(* PLC project Unnamed, Unknown Unnamed 1 *)
(* stored: creationDateTime 2025-10-22T19:37:31, modificationDateTime 2025-10-29T13:50:30 *)

PROGRAM plc_controller
  VAR
    In_Start_Stop AT %IX100.2 : BOOL;
    In_Temp_Up AT %IX100.0 : BOOL;
    In_Temp_Down AT %IX100.1 : BOOL;
    In_Emergency_Stop AT %IX100.3 : BOOL;
    Out_Status_LED AT %QX100.7 : BOOL;
    Out_Display_LED0 AT %QX100.6 : BOOL;
    Out_Display_LED1 AT %QX100.5 : BOOL;
    Out_Display_LED2 AT %QX100.4 : BOOL;
    Out_Display_LED3 AT %QX100.3 : BOOL;
    Out_Display_LED4 AT %QX100.2 : BOOL;
    Out_Display_LED5 AT %QX100.1 : BOOL;
  END_VAR
  VAR
    Out_Servo_PWM_Chann : SINT := 1;
    Servo_Freq : REAL := 50.0;
    Servo_Angle : REAL := 0.0;
    Heating_On : BOOL := FALSE;
    Element_On : BOOL := FALSE;
    Emergency_Stop : BOOL;
    Global_Enable : BOOL;
    Display_Index : INT := 0;
    Temp_Setting : INT := 0;
    Temperature : REAL;
    MAX_TEMP_SETTING : INT := 10;  (* CONSTANT describes the maximum temperature setting *)
    R_TRIG0 : R_TRIG;
    CTUD0 : CTUD;
    TON0 : TON;
    R_TRIG1 : R_TRIG;
    CTUD1 : CTUD;
    PID0 : PID;
    TON1 : TON;
    R_TRIG2 : R_TRIG;
    R_TRIG3 : R_TRIG;
  END_VAR
  VAR  (* added by the conversion: wires and edge detectors of the diagram *)
    _NOT21_OUT : BOOL;
    R_TRIG1_2 : R_TRIG;
    R_TRIG2_2 : R_TRIG;
    R_TRIG3_2 : R_TRIG;
    R_TRIG4 : R_TRIG;
    _MUL240_OUT : REAL;
  END_VAR

(* FBD diagram, written out as Structured Text *)
(* Heating on/off toggle functionality *)
(* Simple heating simulation *)
(* Multiply counter output, and add room temperature. *)
(* Emergency Stop *)
(* Temperature setting controls *)
(* Change display index in set mode *)
_NOT21_OUT := NOT Heating_On;
R_TRIG1_2(CLK := NOT CTUD0.QU AND In_Temp_Up AND _NOT21_OUT);
R_TRIG2_2(CLK := In_Temp_Down AND _NOT21_OUT AND NOT CTUD0.QD);
CTUD0(CU := R_TRIG1_2.Q, CD := R_TRIG2_2.Q, PV := MAX_TEMP_SETTING);
Temp_Setting := CTUD0.CV;
R_TRIG0(CLK := In_Start_Stop);
Heating_On := (R_TRIG0.Q XOR Heating_On) AND Global_Enable;
Out_Status_LED := Heating_On;
(* Change display index in set heating mode *)
(* Display temperature setting *)
Out_Display_LED0 := Display_Index = 0 OR Display_Index = 1;
Out_Display_LED3 := Display_Index = 5 OR Display_Index = 6 OR Display_Index = 7;
(* PID Control Loop
- P = -0.5
- I = 1000.0
- D = 0.5 *)
Out_Display_LED1 := Display_Index = 1 OR Display_Index = 2 OR Display_Index = 3;
Out_Display_LED4 := Display_Index = 7 OR Display_Index = 8 OR Display_Index = 9;
Out_Display_LED2 := Display_Index = 3 OR Display_Index = 4 OR Display_Index = 5;
Out_Display_LED5 := Display_Index = 9 OR Display_Index = 10;
TON0(IN := NOT R_TRIG1.Q, PT := T#20ms);
R_TRIG1(CLK := TON0.Q);
R_TRIG3_2(CLK := R_TRIG1.Q AND Element_On);
R_TRIG4(CLK := NOT Element_On AND R_TRIG1.Q);
CTUD1(CU := R_TRIG3_2.Q, CD := R_TRIG4.Q, PV := 1000);
Temperature := INT_TO_REAL(CTUD1.CV) * 0.1 + 60.0;
IF Global_Enable AND NOT Heating_On THEN Display_Index := Temp_Setting; END_IF;
IF Heating_On THEN Display_Index := LIMIT(0, REAL_TO_INT((Temperature - 80.0) / 100.0 * INT_TO_REAL(MAX_TEMP_SETTING)), MAX_TEMP_SETTING); END_IF;
PID0(AUTO := TRUE, PV := Temperature, SP := INT_TO_REAL(Temp_Setting * 10 + 80), KP := -0.5, TR := 1000.0, TD := 0.5, CYCLE := T#20ms);
Element_On := Heating_On AND REAL_TO_BOOL(LIMIT(0.0, PID0.XOUT, 1.0));
(* Servo valve controls
CHANNEL = 0 for %QW0
FREQ = 50Hz *)
TON1(IN := NOT R_TRIG2.Q, PT := T#100ms);
R_TRIG2(CLK := TON1.Q);
IF R_TRIG2.Q THEN Servo_Angle := LIMIT(0.0, SEL(NOT Heating_On, Servo_Angle + 1.8, Servo_Angle - 1.8), 144.0); END_IF;
R_TRIG3(CLK := In_Emergency_Stop);
Emergency_Stop := R_TRIG3.Q XOR Emergency_Stop;
Global_Enable := NOT Emergency_Stop;
IF NOT Global_Enable THEN Display_Index := -1; END_IF;
_MUL240_OUT := (Servo_Angle / 90.0 + 0.5) / (1000.0 / Servo_Freq) * 100.0;
(* drawn but not wired to any output: Out_Servo_PWM_Chann, Servo_Freq *)
END_PROGRAM

CONFIGURATION Config0
  RESOURCE Res0 ON PLC
    TASK task0(INTERVAL := T#20ms, PRIORITY := 0);
    PROGRAM instance0 WITH task0 : plc_controller;
  END_RESOURCE
END_CONFIGURATION
